// TIA Portal V19 export
DATA_BLOCK "PPrgArchive1"   // DB501
// stored: IsOnlyStoredInLoadMemory true, MemoryReserve 0, Namespace G
   VAR RETAIN
      PRG : Array[1..100] of "PPrg_Data";
   END_VAR
BEGIN
   PRG[1].Header.PrgNo := 123;
   PRG[2].Header.PrgNo := 67;
   PRG[3].Header.PrgNo := 300;
   PRG[4].Header.PrgNo := 150;
   PRG[5..6].Header.PrgNo := 0;
   PRG[7].Header.PrgNo := 299;
   PRG[8].Header.PrgNo := 1;
   PRG[1].Header.PrgName := 'copy of adasdasd';
   PRG[2].Header.PrgName := 'copy of pippo';
   PRG[3].Header.PrgName := 'copy of adasdasd';
   PRG[4].Header.PrgName := 'SONO LO SCADA';
   PRG[5..6].Header.PrgName := '';
   PRG[7].Header.PrgName := 'adasdasd';
   PRG[8].Header.PrgName := 'New empty program';
END_DATA_BLOCK
